FUNCTION_BLOCK FB_QuantityLREALPublicMock EXTENDS FB_FalliblePublicMock IMPLEMENTS I_QuantityLREALPublic
VAR
    fValue : LREAL;
    sUnits : T_MaxString;
END_VAR


METHOD Copy
VAR_INPUT
    QuantityToCopy : I_QuantityLREAL;
END_VAR

Val := QuantityToCopy.Val;
Units := QuantityToCopy.Units;

IF QuantityToCopy.GetError() THEN
    SetError(Msg := QuantityToCopy.GetErrorMsg());
ELSE
    ClearError();
END_IF
END_METHOD


METHOD Equals : BOOL
VAR_INPUT
    Quantity	: I_QuantityLREAL;
END_VAR

Equals := Quantity.Units = Units AND Quantity.Val = Val;
END_METHOD


PROPERTY Units : T_MaxString
GET

Units := sUnits;
END_GET
SET

sUnits := Units;
END_SET
END_PROPERTY


PROPERTY Val : LREAL
GET

Val := fValue;
END_GET
SET

fValue := Val;
END_SET
END_PROPERTY

END_FUNCTION_BLOCK

(* stored: Version 1.1.0.1
   POU FB_QuantityLREALPublicMock: Id {d5300c7f-6e41-485a-a6c7-fc4dd72da079}, SpecialFunc None
   Method Copy: Id {31bab2b9-47f7-4b43-9ab9-4e60f984e71c}
   Method Equals: Id {3b86ff3d-71a5-44c1-a6f9-6ea99eabbd7c}
   Property Units: Id {992c7fcd-f7ab-4268-92a3-a2302b5f867b}
   Get Get: Id {cd4060b6-cc83-4d01-be92-70f0f47259f2}
   Set Set: Id {847cfcfb-8246-447f-afbe-2dfd62ac3403}
   Property Val: Id {5ae91315-6597-48d9-9fb9-751cfc9d19fa}
   Get Get: Id {52a853f1-b2bd-46dd-90c4-a0e53f90d5b1}
   Set Set: Id {b9399bb7-49e6-40ee-858e-a36815fbd8e8} *)
